FUNCTION_BLOCK I_RHS (* Primary or Rear Hitch Status RHS *)
  (* Standard: ISO 11783-7; Classification: PGN 65093; Function: Primary or Rear Hitch Status RHS; Description: Copyright (c) 2024 HR Agrartechnik GmbH This program and the accompanying materials are made available under the terms of the Eclipse Public License 2.0 which is available at https://www.eclipse.org/legal/epl-2.0/ SPDX-License-Identifier: EPL-2.0 Message that provides the measurement of the current rear-hitch parameters. https://docs.ms-muc-docs.de/projects/isobus-other-docs/de/latest/PGN/PGN_65093.html *)
  (* Version 1.0, 2024-07-09, Franz Hoepfinger, HR Agrartechnik GmbH *)
  PACKAGE isobus::tecu;
  IMPORT eclipse4diac::core::TypeHash;
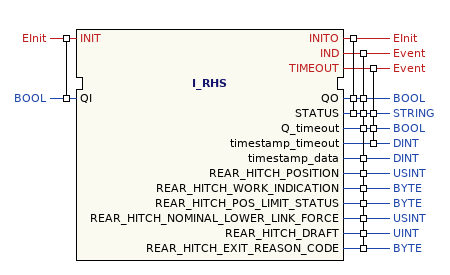
  EVENT_INPUT
    INIT : EInit WITH QI; (* Service Initialization *)
  END_EVENT
  EVENT_OUTPUT
    INITO : EInit WITH QO, STATUS; (* Initialization Confirm *)
    IND WITH QO, timestamp_data, STATUS, Q_timeout, REAR_HITCH_POSITION, REAR_HITCH_WORK_INDICATION, REAR_HITCH_POS_LIMIT_STATUS, REAR_HITCH_NOMINAL_LOWER_LINK_FORCE, REAR_HITCH_DRAFT, REAR_HITCH_EXIT_REASON_CODE; (* Indication from Resource *)
    TIMEOUT WITH timestamp_timeout, STATUS, Q_timeout;
  END_EVENT
  VAR_INPUT
    QI : BOOL; (* Event Input Qualifier *)
  END_VAR
  VAR_OUTPUT
    QO : BOOL; (* Event Output Qualifier *)
    STATUS : STRING;
    Q_timeout : BOOL;
    timestamp_timeout : DINT;
    timestamp_data : DINT;
    REAR_HITCH_POSITION : USINT; (* Rear Hitch Position (see Attributes for Details) *) {SET_ATTRIBUTE(SPN, 1873)} {SET_ATTRIBUTE(SP_Name, 'Rear Hitch Position')} {SET_ATTRIBUTE(SP_Position_In_PG, '1')} {SET_ATTRIBUTE(SP_Length, 8)} (* 8 bits *) {SET_ATTRIBUTE(Scaling, '0.4 %/bit')} {SET_ATTRIBUTE(Offset, )} {SET_ATTRIBUTE(Link, 'https://docs.ms-muc-docs.de/projects/isobus-other-docs/de/latest/PGN/PGN_65093.html#spn-1873-rear-hitch-position')}
    REAR_HITCH_WORK_INDICATION : BYTE; (* Rear Hitch In-work Indication *) {SET_ATTRIBUTE(SPN, 1877)} {SET_ATTRIBUTE(SP_Name, 'Rear Hitch In-work Indication')} {SET_ATTRIBUTE(SP_Position_In_PG, '2.7')} {SET_ATTRIBUTE(SP_Length, 2)} (* 2 bits *) {SET_ATTRIBUTE(Scaling, '4 states/2 bit')} {SET_ATTRIBUTE(Offset, )} {SET_ATTRIBUTE(Link, 'https://docs.ms-muc-docs.de/projects/isobus-other-docs/de/latest/PGN/PGN_65093.html#spn-1877-rear-hitch-in-work-indication')}
    REAR_HITCH_POS_LIMIT_STATUS : BYTE; (* Rear Hitch Position Limit status *) {SET_ATTRIBUTE(SPN, 5151)} {SET_ATTRIBUTE(SP_Name, 'Rear Hitch Position Limit status')} {SET_ATTRIBUTE(SP_Position_In_PG, '2.4')} {SET_ATTRIBUTE(SP_Length, 3)} (* 3 bits *) {SET_ATTRIBUTE(Scaling, '8 states/3 bit')} {SET_ATTRIBUTE(Offset, )} {SET_ATTRIBUTE(Link, 'https://docs.ms-muc-docs.de/projects/isobus-other-docs/de/latest/PGN/PGN_65093.html#spn-5151-rear-hitch-position-limit-status')}
    REAR_HITCH_NOMINAL_LOWER_LINK_FORCE : USINT; (* Rear Nominal Lower Link Force *) {SET_ATTRIBUTE(SPN, 1881)} {SET_ATTRIBUTE(SP_Name, 'Rear Nominal Lower Link Force')} {SET_ATTRIBUTE(SP_Position_In_PG, '3')} {SET_ATTRIBUTE(SP_Length, 8)} (* 8 bits *) {SET_ATTRIBUTE(Scaling, '0.8 %/bit')} {SET_ATTRIBUTE(Offset, -100)} {SET_ATTRIBUTE(Link, 'https://docs.ms-muc-docs.de/projects/isobus-other-docs/de/latest/PGN/PGN_65093.html#spn-5151-rear-hitch-position-limit-status')}
    REAR_HITCH_DRAFT : UINT; (* Rear Draft *) {SET_ATTRIBUTE(SPN, 1879)} {SET_ATTRIBUTE(SP_Name, 'Rear Draft')} {SET_ATTRIBUTE(SP_Position_In_PG, '4-5')} {SET_ATTRIBUTE(SP_Length, 16)} (* 16 bits *) {SET_ATTRIBUTE(Scaling, '10 N/bit')} {SET_ATTRIBUTE(Offset, -320000)} {SET_ATTRIBUTE(Link, 'https://docs.ms-muc-docs.de/projects/isobus-other-docs/de/latest/PGN/PGN_65093.html#spn-1879-rear-draft')}
    REAR_HITCH_EXIT_REASON_CODE : BYTE; (* Rear hitch exit/reason code *) {SET_ATTRIBUTE(SPN, 5819)} {SET_ATTRIBUTE(SP_Name, 'Rear hitch exit/reason code')} {SET_ATTRIBUTE(SP_Position_In_PG, '6.1')} {SET_ATTRIBUTE(SP_Length, 6)} (* 6 bits *) {SET_ATTRIBUTE(Scaling, '64 states/6 bit')} {SET_ATTRIBUTE(Offset, )} {SET_ATTRIBUTE(Link, 'https://docs.ms-muc-docs.de/projects/isobus-other-docs/de/latest/PGN/PGN_65093.html#spn-5819-rear-hitch-exit-reason-code')}
  END_VAR
END_FUNCTION_BLOCK
